// TIA Portal V19 export
TYPE "C701_VAR_IF_KOKR_TYPIC"
   STRUCT
      STO { ExternalAccessible := 'False'; ExternalVisible := 'False'; ExternalWritable := 'False'} : Struct   // Opsomming van alle storingen
         A001 : Bool;   // Storing van de motorbeveiliging van pomp 1
         A002 : Bool;   // Storing van de motorbeveiliging van pomp 2
         A003 : Bool;   // Fout temperatuurmeting vertrek
         A004 : Bool;   // Fout temperatuurmeting retour
         A005 : Bool;   // Fout drukmeting
      END_STRUCT;
   END_STRUCT;
END_TYPE
